{attribute addProperty BoxType "KL9976-0050"}
{attribute addProperty Id "Channel_100"}
{attribute addProperty CRC "3630262351"}
{attribute addProperty SizeInBites "0"}
{attribute addProperty SizeInBytes "0"}
TYPE KL_D861684F :
STRUCT
	{attribute addProperty Name "Channel_1"}
	Channel_1 : ;
END_STRUCT
END_TYPE

(* stored: Version 1.2.0.0, ProductVersion 3.1.4024.9
   DUT KL_D861684F: Id {5057d2e7-1bf0-41c6-aaa6-b42162f6e583} *)
